FUNCTION_BLOCK FB_WorkerDefGrid_Camera EXTENDS FB_WorkerDefGrid IMPLEMENTS I_CameraSink
VAR
  // references
  _pAdsCam        : POINTER TO ST_ADS_CAMERA;
  _iParamMediator : I_ParamMediator;
  
  // camera list
  _iCamList       : ARRAY[1..nMAXCAM] OF I_Camera; 
  _sCamName       : ARRAY[1..5] OF STRING;
  _nRegisteredCam : UDINT;    // number registered cameras
  _iActiveCam     : I_Camera; // active selected camera interface
  
  // cam status
  _bCamValid      : BOOL;
  _bCamReady      : BOOL;    // Camera no error
  _bConnectionOk  : BOOL;    //
  _bTeachOk       : BOOL;    // Teach successful
  _nTeachedPoints : UDINT;   // Teached points for this job
  _nScannedPoints : UDINT;   // Scanned points on current sheet
  _bCamStarted    : BOOL;    // Camera started
  _bCamDone       : BOOL;    // Camera done
  _nAddedPoint    : UDINT;   // Added point to image deformation
 
  _bLineCamType   : BOOL;    // TRUE if it's a LineCamera
  _bSetInitCam    : BOOL;    // set initial camera
  
  // deformation status
  _eDeformStep                : E_DeformationStep;   // status deformation of ct
  
  // Messages
  _pMsgConfig                   : POINTER TO ST_MSG_CONFIG;
  bCamNotAvailable             : BOOL;
  fbMsg_CamNotAvailable        : FB_MESSAGE;
  bCamModeNotSupported         : BOOL;
  fbMsg_CamModeNotSupported    : FB_MESSAGE;
  fbMsg_CamNoConnection        : FB_MESSAGE;
  
END_VAR

VAR PERSISTENT
  _fFeatureGrid   : LREAL := 2048;  // feature grid witdh (feature pich in x of cam frames)
  _nActiveCam     : UDINT := 1;     // active camera selection
END_VAR

VAR CONSTANT
  nMAXCAM : UDINT := 5;
END_VAR

METHOD PRIVATE ActivateCamera : BOOL
VAR_INPUT
  iCam : I_Camera;
END_VAR
VAR
  i : UDINT;
END_VAR
IF iCam = 0 THEN F_Report_Error(ErrType:=EN_REPORT_ERROR_TYPE.Report_Error_0Pointer); RETURN; END_IF

IF _iActiveCam <> 0 THEN // Remove existing links
  _iActiveCam.DeactivateCam(iSink := THIS^);
END_IF

IF iCam.ActivateCam(iCameraSink := THIS^) THEN
  // get and set array index of registered cameras 
  FOR i :=1 TO _nRegisteredCam DO
    IF iCam = _iCamList[i] THEN
      _nActiveCam := i;              // set array index for visu/drop down
      EXIT; // select first found cam
    END_IF
  END_FOR
  _iActiveCam := iCam;        // set new cam
  ActivateCamera:=TRUE;
ELSE
  ActivateCamera:=FALSE;
END_IF
END_METHOD

METHOD AddCamPoint : BOOL
VAR_INPUT
	sDeformationPoint	: ST_DeformationPointAccurate;
END_VAR
{warning 'TODO: add a small queue for input points'}

IF _pAttachedCt <> 0 THEN //Container attached?
  AddCamPoint := _pAttachedCt^.AddCamPoint(sPoint:=sDeformationPoint);
  IF AddCamPoint THEN 
    _nAddedPoint :=_nAddedPoint+1;
    //cameraImgProc(newDeformationPoint:=iDeformationPoint);  //Update image processing
  ELSE
    LogError(Msg:='addCamPoint failed, add to CT error');
  END_IF;
ELSE
  LogWarning(Msg:=F_Concat2('addCamPoint failed, no CT attached: ', F_DeformationPointAcc_ToString(sPointAcc:=sDeformationPoint)));
END_IF
END_METHOD

METHOD AddTeachPoint : BOOL
VAR_INPUT
	sTeachPoint	: ST_DeformationPointAccurate;
END_VAR

// ignore the teach points for now
END_METHOD

METHOD PROTECTED  Attach : BOOL
VAR_INPUT
  iCT              : I_CT;                         (*container at triggered event position*)
END_VAR
VAR
  tempCt :  POINTER TO FB_ContainerDefGrid;
  bDeformErr : BOOL;
  eDeformStep : E_DeformationStep;
END_VAR
Attach := FALSE;
IF SUPER^.Attach(iCT:=iCT) THEN
  // OK, attached (enabled, was ok to be attached)
  
  bDeformErr := _pAttachedCt^.getDeformationStatus(eDStep=>eDeformStep);   // get latest status 
  
  // Additional worker checks

  // - deformation started? and no deformation error so far
  IF bDeformErr OR eDeformStep = E_DeformationStep.nothing THEN
    Release(iCT:=iCT);  // nothing to do anymore

  // - job is valid?
  ELSIF _pAttachedCt^.pJob = 0 OR NOT _bJobActive THEN
    _pAttachedCt^.AbortDeformation(sReason:='No valid job', Src:=_pEcSrc^);
    Release(iCT:=iCT);
       
  // - camera ready
  ELSIF (NOT _bCamValid OR NOT _bCamReady) THEN  // check if cam is ready
    _pAttachedCt^.AbortDeformation(sReason:='Camera invalid or not ready for attach', Src:=_pEcSrc^);
    Release(iCT:=iCT);
  
  // OK attach
  ELSE
    Attach := TRUE;
	END_IF
  
  //Reset image processing
  _nAddedPoint := 0;
  _nScannedPoints := 0;

ELSE
  // parent attach failed case
END_IF
END_METHOD

PROPERTY bCamOk : BOOL
GET
bCamOk := _bCamValid;
END_GET
END_PROPERTY

PROPERTY bConnError : BOOL
GET
// TODO: propose the communication error on a better way.
bConnError := NOT _bConnectionOk;
END_GET
END_PROPERTY

PROPERTY bLineCamActive : BOOL
GET
bLineCamActive := _bLineCamType;
END_GET
END_PROPERTY

PROPERTY fCameraToPrintOffset : LREAL
GET
IF _iActiveCam <> 0 THEN
  fCameraToPrintOffset := _iActiveCam.fCameraToPrintOffset;
END_IF
END_GET
END_PROPERTY

PROPERTY fDetectToCamOffset : LREAL
GET
IF _iActiveCam <> 0 THEN
  fDetectToCamOffset := _iActiveCam.fDetectToCameraOffset;
END_IF
END_GET
END_PROPERTY

METHOD Init
VAR_INPUT
  iWorkerParams : I_WorkerParams;
  pMsgConfig : POINTER TO ST_MSG_CONFIG;         // message config
  fPrintResolution : LREAL := 1;                 // print(head) resolution in [dpi]
  fSubPxResolution : LREAL := 1;                 // SubPixel resolution [SubPx], resolution factor (fI_PrintResolution*fI_SubPxResolution=>Output resolution)
END_VAR
VAR
  lCtr : UDINT;
END_VAR
SUPER^.Init(iWorkerParams:=iWorkerParams, pMsgConfig:=pMsgConfig, fPrintResolution:=fPrintResolution, fSubPxResolution:=fSubPxResolution);

IF pMsgConfig = 0 THEN LogError('Init: invalid message config given'); END_IF 

(*Messaging*)
_pMsgConfig := pMsgConfig;

fbMsg_CamNotAvailable.pI_MsgConfig := _pMsgConfig;
fbMsg_CamNotAvailable.iI_MsgLocation := ePr_BLK_CAMERA;
fbMsg_CamNotAvailable.iI_MsgNumber := eC_DMAX_CAM_NOTAVAIL;

fbMsg_CamModeNotSupported.pI_MsgConfig := _pMsgConfig;
fbMsg_CamModeNotSupported.iI_MsgLocation := ePr_BLK_CAMERA;
fbMsg_CamModeNotSupported.iI_MsgNumber := eC_DMAX_CAM_MODE_NOTSUPPORTED; // camera not available

fbMsg_CamNoConnection.pI_MsgConfig := _pMsgConfig;
fbMsg_CamNoConnection.iI_MsgLocation := ePr_BLK_CAMERA;
fbMsg_CamNoConnection.iI_MsgNumber := eCMa_TCPIP_COMM_ERROR;    // tcpip connection error

_bConnectionOk := TRUE;
_bSetInitCam := TRUE; // request a default camera
END_METHOD

METHOD InitWorkerCamera
VAR_INPUT
  pAdsIf  : POINTER TO ST_ADS_CAMERA;
  iDefGridParamMediator : I_ParamMediator;
END_VAR
IF NOT bInitialized OR _iWorkerParams.pCTManager = 0 THEN LogError('Base Worker not initialized! call init() before'); RETURN; END_IF
IF pAdsIf = 0 THEN bInitialized := FALSE; LogError('Invalid parameter, no valid ads interface camera'); RETURN; END_IF
IF iDefGridParamMediator = 0 THEN bInitialized := FALSE; LogError('Invalid parameter, no valid param mediator'); RETURN; END_IF

_pAdsCam := pAdsIf;
_iParamMediator := iDefGridParamMediator;
END_METHOD

METHOD PRIVATE is_linecam : BOOL
VAR_INPUT
  sCamName : STRING;
END_VAR
is_linecam := SEL(FIND(F_ToLCase(sCamName), 'linecam') > 0, FALSE, TRUE);  // is it a LineCamera?
END_METHOD

METHOD   mJobStart
VAR_INPUT
	sJobDef	: CalmarCompPrint.I_JobDefinition;
END_VAR
VAR
  iNewCam : I_Camera;
END_VAR
IF _pAdsCam <> 0 THEN

  bCamNotAvailable := FALSE;
  bCamModeNotSupported := FALSE;

  // activate matching camera
  iNewCam := selectCamera(eNewCam:=_pAdsCam^.eI_CameraDevice);    // get camera settings from ADS
  IF NOT ActivateCamera(iCam:=iNewCam) THEN
    LogError(F_Concat2('Could not activate camera: ', TO_STRING(_pAdsCam^.eI_CameraDevice)));
    bCamNotAvailable := TRUE;
  ELSE
    // config camera from job
    _iActiveCam.fSubstrateLength := sJobDef.fSubstrateDepth;      // [m]
    _iActiveCam.fSubstrateWidth  := sJobDef.fSubstrateWidth;      // [m]
    _iActiveCam.fImageLength     := sJobDef.fImageDepth  / 1000;  // [mm] -> [m]
    _iActiveCam.fImageWidth      := sJobDef.fImageWidth  / 1000;  // [mm] -> [m]
    _iActiveCam.fFrameLength     := _fFeatureGrid;                // [px]
    bCamModeNotSupported := NOT _iActiveCam.setCameraMode(eCameraMode := _pAdsCam^.eI_CameraMode);     // set camera mode
    _iActiveCam.bEnableTrigger   := TRUE;    
    _iActiveCam.bManualTeach     := FALSE;
    _iActiveCam.mJobStart();

    // check settings
    IF _iActiveCam.fSubstrateLength = 0 THEN LogError('mJobStart() invalid SubstrateLength'); END_IF
    IF _iActiveCam.fSubstrateWidth = 0 THEN LogError('mJobStart() invalid SubstrateWidth'); END_IF
    IF _iActiveCam.fImageLength = 0 THEN LogError('mJobStart() invalid ImageLength'); END_IF
    IF _iActiveCam.fImageWidth = 0 THEN LogError('mJobStart() invalid ImageWidth'); END_IF
    
    // special case
    _bLineCamType := is_linecam(_iActiveCam.sName);  // is it a LineCamera?
  END_IF
END_IF

_bJobActive := TRUE;
END_METHOD

METHOD  mJobStop
VAR_INPUT
	sStatus	: CalmarCompPrint.I_JobStatus;
END_VAR
_bJobActive := FALSE;
END_METHOD

METHOD RegisterCamera : BOOL
VAR_INPUT
  iNewCam : I_Camera;
END_VAR
IF _nRegisteredCam < nMAXCAM AND iNewCam <> 0 THEN
  // configure message interface
  iNewCam.setMsgInterface(pMsgConfig:=_pMsgConfig);     // set message interface
  // add to internal list
  _nRegisteredCam := _nRegisteredCam + 1;
  _iCamList[_nRegisteredCam] := iNewCam;
  _sCamName[_nRegisteredCam] := iNewCam.sName;
  RegisterCamera := TRUE;
END_IF
END_METHOD

METHOD PRIVATE reviewState : BOOL
VAR
  bModeLowerThanRequested       : BOOL;
END_VAR
// review all camera states and set messages accordingly
IF _bJobActive AND _iActiveCam <> 0 THEN

  // -> mode less than desired
  IF _pAdsCam^.eI_CameraMode < _iActiveCam.eCameraMode THEN
    bModeLowerThanRequested := TRUE;
  END_IF

ELSE
  ;
END_IF
END_METHOD

PROPERTY sCameraGridSettings : ST_CameraGridSettings
GET
sCameraGridSettings.bValid := _bCamValid;
IF _bCamValid THEN
  sCameraGridSettings.eCameraMode := SEL(_iActiveCam<>0, E_CameraMode.NoCorrection, _iActiveCam.eCameraMode);
  sCameraGridSettings.fGridFeaturePitch := _fFeatureGrid;
END_IF
END_GET
END_PROPERTY

(*
  Select a registered camera from the requested device type.
*)
METHOD PRIVATE selectCamera : I_Camera
VAR_INPUT
  eNewCam  : E_CameraDevice;      // requested camera type
END_VAR
VAR
  bFound : BOOL;
  i : UDINT;
  sOld, sNew : STRING :='';
END_VAR
// select related camera (choose first matching)
bFound := FALSE;
FOR i :=1 TO _nRegisteredCam DO
  IF eNewCam = _iCamList[i].eDeviceType THEN
    // found
    selectCamera  := _iCamList[i]; // select new cam
    bFound := TRUE;
    EXIT; // select first found cam
	END_IF
END_FOR

IF NOT bFound THEN
  IF _iActiveCam <> 0 THEN sOld := _iActiveCam.sName; END_IF
  IF _pAdsCam <> 0 THEN sNew := TO_STRING(_pAdsCam^.eI_CameraDevice); END_IF
  
  LogError(F_Concat4('Unavailable camera selected=', sNew, ', use cam=', sOld));
  selectCamera  := _iActiveCam; // return camera to before
END_IF
END_METHOD

METHOD setManualTeach
VAR_INPUT
  eCameraDevice    : E_CameraDevice;  
  fSubstrateLength : LREAL;   // teach substrate length
  fSubstrateWidth  : LREAL;   // teach substrate width
END_VAR
VAR
  iNewCam : I_Camera;
END_VAR
// activate Camera

iNewCam := selectCamera(eNewCam:=eCameraDevice);    // Scanner
IF NOT ActivateCamera(iCam:=iNewCam) THEN
  LogError(F_Concat2('Could not activate camera: ', TO_STRING(eCameraDevice)));
ELSE
  // config camera from manual teach
  _iActiveCam.fSubstrateLength := fSubstrateLength;
  _iActiveCam.fSubstrateWidth  := fSubstrateWidth;
  _iActiveCam.fImageLength     := fSubstrateLength;
  _iActiveCam.fImageWidth      := fSubstrateWidth;
  _iActiveCam.setCameraMode(eCameraMode :=E_CameraMode.Auto);     // set camera mode
  _iActiveCam.bEnableTrigger   := TRUE;   // enables trigger in CameraTrigger
  _iActiveCam.bManualTeach     := TRUE;   // enables manual trigger mode in CameraTrigger
  
  // special case
  _bLineCamType := is_linecam(_iActiveCam.sName);  // is it a LineCamera?
END_IF
END_METHOD

METHOD  work
VAR_INST
  rT_CamStarted : R_TRIG;
  rT_CamDone : R_TRIG;
  bReqToStartCamOnCt : BOOL;
END_VAR
VAR
  lCtr : UDINT;
END_VAR
IF _iParamMediator = 0 THEN RETURN; END_IF

SUPER^.work();

//-----------------------------------------------------------
//- automatic worker setup & control
IF _bSetInitCam AND _iActiveCam = 0 THEN    // try to set a default camera at start
  ActivateCamera(selectCamera(eNewCam:=E_CameraDevice.SheetDetect));
  _bSetInitCam := FALSE;
  _bCamValid := TRUE;
ELSIF _iActiveCam <> 0 THEN                 // a camera is activated
  
  // --- cyclic call always when cam is active ---
  _bCamValid := TRUE;
  //-- update status  
  _bCamReady := _iActiveCam.GetCamStatus(
                              bConnectionOK => _bConnectionOk, 
                              bTeachOk => _bTeachOk, 
                              nTeachedPoints => _nTeachedPoints, 
                              nScannedPoints => _nScannedPoints,
                              bCamStarted => _bCamStarted,
                              bCamDone => _bCamDone);
  // -- worker position setup
  IF _pAttachedCt = 0 THEN     // Update only without attached container
    // WorkerPosition 
    fPosition := fDetectToCamOffset;
  END_IF
ELSE
  _bCamValid := FALSE;                    // invalid camera
END_IF
rT_CamStarted(CLK:=_bCamStarted);
IF rT_CamStarted.Q THEN bReqToStartCamOnCt := TRUE; END_IF
rT_CamDone(CLK:=_bCamDone); 


// -----------------------------------------------------------
// Work only with attached container
IF _pAttachedCt <> 0 THEN
  bError := _pAttachedCt^.getDeformationStatus(eDStep => _eDeformStep);
  
  IF _eDeformStep > E_DeformationStep.nothing AND _bCamReady AND _bTeachOk THEN      // start only if py started
    IF bReqToStartCamOnCt THEN
      // -- setup deformation with cam settings
      LogLvl(Lvl:=E_LogSeverity.Debug, Msg:=F_Concat2('CamStarted mode: ', TO_STRING(_iActiveCam.eCameraMode)));
      _pAttachedCt^.StartCamera(eCameraMode:=_iActiveCam.eCameraMode, fFeatureGrid:=_fFeatureGrid);
      bReqToStartCamOnCt := FALSE; // reset
		END_IF
    IF _bCamDone AND _eDeformStep >= E_DeformationStep.cameraStarted THEN
        LogLvl(Lvl:=E_LogSeverity.Debug, Msg:='CamDone');
        Release(_pAttachedCt^);
    END_IF
      
    (*IF _eDeformStep >= E_DeformationStep.cameraStarted AND _nScannedPoints > 3 THEN   // TODO: handle this in py script / select local Grid generation or script
      _pAttachedCt^.UpdateDeformation();         // update with cam feature grid  
      IF _bCamDone THEN
        Release(_pAttachedCt^);
      END_IF
    END_IF*)
    
    
  ELSE
    IF _bCamStarted THEN
      LogLvl(Lvl:=E_LogSeverity.Debug, Msg:=F_Concat6('CamDone step: ', TO_STRING(_eDeformStep), ' CamReady: ', TO_STRING(_bCamReady), ' TeachOk: ', TO_STRING(_bTeachOk)));
      Release(_pAttachedCt^);
    END_IF
  END_IF
END_IF

// call messages
fbMsg_CamNotAvailable    (bI_Status:=bCamNotAvailable);
fbMsg_CamModeNotSupported(bI_Status:=bCamModeNotSupported);
fbMsg_CamNoConnection    (bI_Status:=bConnError);
END_METHOD

END_FUNCTION_BLOCK

(* stored: Version 1.1.0.1, ProductVersion 3.1.4024.11
   POU FB_WorkerDefGrid_Camera: Id {6056a89a-8aeb-47d0-8a92-08f600f3d0b4}, SpecialFunc None
   Folder I_CameraSink: Id {9ec3d051-264b-49d1-b711-6f2c7c383bca}
   Folder I_PrintStatusClient: Id {1c674285-cbe4-4e1b-ab1f-c86c3f21aeed}
   Method ActivateCamera: Id {99a01e14-fa02-42f4-a663-cfcdcb61b4bd}
   Method AddCamPoint: Id {f453464a-4078-41ca-a01d-17dc87f686bd}
   Method AddTeachPoint: Id {f2606cab-e071-41ba-b4be-aa219442a713}
   Method Attach: Id {af64d5ac-9c9c-46b2-994b-9271d2dee30d}
   Property bCamOk: Id {5ecde9b0-3187-4838-9771-10aabc571882}
   Get Get: Id {a8d145ae-a852-4e60-a712-39a8f1889f94}
   Property bConnError: Id {134a7455-f42f-4d23-9774-a052257145a6}
   Get Get: Id {923e802f-8818-4054-aa36-ae56db26c1db}
   Property bLineCamActive: Id {76835a52-9212-491e-85d8-29398d3bbb8a}
   Get Get: Id {dfd3a19d-9364-487f-af97-eece4f64fd7b}
   Property fCameraToPrintOffset: Id {c7f93a14-f1d1-4c31-a277-d18b12fc9117}
   Get Get: Id {7463415f-08fd-4759-a1b6-38cdc37fe30e}
   Property fDetectToCamOffset: Id {65907cba-8221-4545-9cde-7be24c978514}
   Get Get: Id {b606aab6-d61a-48fb-b789-a7a91f4dddeb}
   Method Init: Id {476974fc-f01a-47ef-80b5-8dcae46aef5e}
   Method InitWorkerCamera: Id {d420bbaf-dc4a-4caf-9bae-af7a97686b3a}
   Method is_linecam: Id {75d58c77-ff64-480b-987c-b901e93de9a9}
   Method mJobStart: Id {333f8056-01ee-443a-9254-a4a08a486903}
   Method mJobStop: Id {113ca763-e1d2-471f-992c-fa941c7af403}
   Method RegisterCamera: Id {b220f8fd-cae6-44e9-b212-d3281862fb7a}
   Method reviewState: Id {202e01c9-d11c-44dc-96a6-afdbd379bab6}
   Property sCameraGridSettings: Id {a50fda04-430c-4b45-a5d1-808b5d907b05}
   Get Get: Id {a97a3e24-418c-4e49-a9d0-b9786579a0f4}
   Method selectCamera: Id {68d1de2e-ca32-4101-91d2-cde38cfd0124}
   Method setManualTeach: Id {2e7801cf-e1ac-475d-9d4e-5dbbc1b969bc}
   Method work: Id {51a4cd28-adfd-4791-8e23-e9bc638f5539} *)
